Fanuc KAREL source: kc00003.KL

-- PROVISIONAL review KL for V770-1; original PC SHA256 4f3cb61764bd8813a98199b4a443244367ccc8634c02f45a13427fb5b5e115db
-- Incomplete behavior may be omitted. Consult companion uncertainty JSON. Do not deploy.
PROGRAM KC00003
%NOLOCKGROUP
BEGIN
  -- UNRESOLVED_PC offsets 5-33; opcodes 27,22,22,22,22,31
  -- UNRESOLVED_PC offsets 38-42; opcodes 7F
END KC00003
